Universal Robots PolyScope program: IAC007 Sensors D.urp

Program IAC007 Sensors D (installation=default directory=/programs createdIn=5.9.1.1031110 lastSavedIn=5.9.1.1031110 robotSerialNumber=20195501059)
Calibrated DH parameters: a=[0.000146, -0.418764, -0.053981, 0.000058, -0.000023, 0]; d=[0.162545, 37.319448, -206.067439, 168.881546, 0.09955, 0.099464]; alpha=[1.57004, -0.001979, 0.002304, 1.570607, -1.57066, 0]; deltaTheta=[0, -0.174616, -1.258233, 1.432844, -0.000001, 0]
BeforeStart
  URCap Gripper Activate (Robotiq_Grippers, Robotiq Inc.) dataModel(ResetAndActivateKey=false)
  initial_p := get_actual_tcp_pose()
  MoveJ speed 60 deg/s, acceleration 80 deg/s^2 (useActiveTCP=true) feature=Base
    Waypoint Waypoint (Variable): variable=initial_p
  iac7_dist := 0
  Set DigitalOutput pin=digital_out[1]; digitalValue=0
Robot Program (runOnlyOnce=true)
  URCap Grip Check (Robotiq_Grippers, Robotiq Inc.) dataModel(ObjectDetectedKey=true, DimensionValidationKey=false, DimensionKey=100.0, DimensionDimensionPositiveGapKey=5.0, DimensionNegativeGapKey=5.0, GripperIdKey=1, ModelDefinedKey=true); state(isChildrenLocked=true)
    URCap If (Robotiq_Grippers, Robotiq Inc.)
      Popup Error (haltProgram=false message=Object in gripper. Safe to open? inputType=Text)
      URCap Gripper (Robotiq_Grippers, Robotiq Inc.) dataModel(position=0.0, force=1.0, speed=20.0, positionInDouble=0.0, forceInDouble=1.0, speedInDouble=20.0, slaveIds=[9], blocking=true)
  MoveL speed 250 mm/s, acceleration 1200 mm/s^2 (useActiveTCP=true) feature=Base
    MoveDirectionNode (selectedDirection=ZMinus) feature=Joint_6_name
      Until DISTANCE (allowActions=false deceleration=3 distanceNodeType=STOP) Distance=0.05; motionParameters(blendRadius=0)
  URCap Gripper (Robotiq_Grippers, Robotiq Inc.) dataModel(position=100.0, force=100.0, speed=100.0, positionInDouble=100.0, forceInDouble=100.0, speedInDouble=100.0, slaveIds=[9], blocking=true)
  MoveL speed 250 mm/s, acceleration 1200 mm/s^2 (useActiveTCP=true) feature=Base
    Waypoint measure_storage: TCP in base x=365.03 y=-83.332 z=77.503 mm, rx=-2.1824 ry=-2.2597 rz=0.0001 rad; joints [146.247, -99.032, 135.126, -126.082, 270.083, 144.278] deg; TCP offset x=0 y=0 z=174 mm, rx=0 ry=0 rz=0 rad
  Wait Sleep waitTime=2
  iac7_base_dist := iac7_dist
  Loop Forever
    iac7_delta_z := iac7_dist - iac7_base_dist
    If norm(iac7_delta_z) > 0.002
      Script file /programs/IAC007 Move Script.script
        | global iac7_cur_p = get_actual_tcp_pose()
        | global iac7_new_p = iac7_cur_p
        | iac7_new_p[2] = iac7_new_p[2] - iac7_delta_z
        | movel(iac7_new_p, a=0.5)
Thread Thread_1 (runOnlyOnce=false)
  Script file /programs/IAC7 Laser Thread 2.script
    | global iac7_n_readings = 10
    | i = 0
    | sum = 0
    | while i < iac7_n_readings:
    |   r = get_standard_analog_in(0)
    |   sum = sum + r
    |   sleep(0.001)
    |   i = i + 1
    | end
    | 
    | global iac7_reading = sum / iac7_n_readings * 187.5 - 0.700 * sin(d2r(72))
    | global iac7_dist = 0.1 * iac7_reading + 0.9 * iac7_dist
